// TIA Portal project "Perron038 AMR Siemens_2" (V14)

(* hardware
DEVICE "S7-1200 station_1"  S7-1200 Station
   slot 0: "Rack_0"  S7-1200 Rack  Rack  V1.0
   slot 1: "PLC_1"  CPU 1215C DC/DC/DC  6ES7 215-1AG40-0XB0  V4.2
*)

// ===== PLC "PLC_1"  CPU 1215C DC/DC/DC =====

VAR_GLOBAL   // PLC tag table "Default tag table"
   "Axis_1_Pulse" AT %Q0.0 : Bool;
   "Axis_1_Dir" AT %Q0.1 : Bool;
   "Axis_1_EN" AT %Q0.3 : Bool;
   "i_EndStopFWD" AT %I0.0 : Bool;
   "i_EndStopBWD" AT %I0.1 : Bool;
   "i_Switch8" AT %I0.7 : Bool;
   "i_Switch7" AT %I0.6 : Bool;
   "Servo_Pucks_Duration" AT %QW1002 : Int;
   "Servo_Grip_Duration" AT %QW1004 : Int;
   "System_Byte" AT %MB1 : Byte;
   "FirstScan" AT %M1.0 : Bool;
   "DiagStatusUpdate" AT %M1.1 : Bool;
   "AlwaysTRUE" AT %M1.2 : Bool;
   "AlwaysFALSE" AT %M1.3 : Bool;
   "Clock_Byte" AT %MB0 : Byte;
   "Clock_10Hz" AT %M0.0 : Bool;
   "Clock_5Hz" AT %M0.1 : Bool;
   "Clock_2.5Hz" AT %M0.2 : Bool;
   "Clock_2Hz" AT %M0.3 : Bool;
   "Clock_1.25Hz" AT %M0.4 : Bool;
   "Clock_1Hz" AT %M0.5 : Bool;
   "Clock_0.625Hz" AT %M0.6 : Bool;
   "Clock_0.5Hz" AT %M0.7 : Bool;
   "Tag_1" AT %Q0.2 : Bool;
   "Tag_2" AT %Q0.4 : Bool;
   "q_Lift_Up" AT %Q0.7 : Bool;
   "q_Lift_Down" AT %Q0.6 : Bool;
   "i_LiftDownStop" AT %I0.2 : Bool;
   "i_LiftHalte1" AT %I0.3 : Bool;
END_VAR

DATA_BLOCK "MotorControl_1_DB"   // DB1
{ S7_Optimized_Access := 'TRUE' }
VERSION : 0.1
// stored: InstanceOfName MotorControl_1
"MotorControl_1"
BEGIN
END_DATA_BLOCK

DATA_BLOCK "Horizontal_Movement_FB_DB"   // DB2
{ S7_Optimized_Access := 'TRUE' }
VERSION : 0.1
// stored: InstanceOfName Horizontal_Movement
"Horizontal_Movement"
BEGIN
END_DATA_BLOCK

DATA_BLOCK "ServoControl_1_DB"   // DB4
{ S7_Optimized_Access := 'TRUE' }
VERSION : 0.1
// stored: InstanceOfName ServoControl_Pucks
"ServoControl_Pucks"
BEGIN
END_DATA_BLOCK

DATA_BLOCK "ServoControl_2_DB"   // DB9
{ S7_Optimized_Access := 'TRUE' }
VERSION : 0.1
// stored: InstanceOfName ServoControl_Gripper
"ServoControl_Gripper"
BEGIN
END_DATA_BLOCK

DATA_BLOCK "DB_ModbusTCP_Connect"   // DB10
{ S7_Optimized_Access := 'TRUE' }
VERSION : 0.1
   VAR
      MBTCPClientRead : TCON_IP_v4;
      MBTCPClientRead_DISCONNECT : Bool;
      MBTCPClientRead_BUSY : Bool;
      MBTCPClientRead_ERROR : Bool;
      MBTCPClientRead_STATUS : Word;
   END_VAR
BEGIN
   MBTCPClientRead.InterfaceId := 64;
   MBTCPClientRead.ID := 16#1;
   MBTCPClientRead.ActiveEstablished := 1;
   MBTCPClientRead.RemoteAddress.ADDR[1] := 16#C0;
   MBTCPClientRead.RemoteAddress.ADDR[2] := 16#A8;
   MBTCPClientRead.RemoteAddress.ADDR[4] := 16#14;
   MBTCPClientRead.RemotePort := 502;
   MBTCPClientRead.LocalPort := 502;
   MBTCPClientRead.RemoteAddress.ADDR[3] := 16#C;
   MBTCPClientRead.ConnectionType := 16#B;
END_DATA_BLOCK

DATA_BLOCK "MBTCP_Data"   // DB11
{ S7_Optimized_Access := 'FALSE' }
VERSION : 0.1
   VAR
      Data : Array[1..1200] of Word;
   END_VAR
BEGIN
END_DATA_BLOCK

DATA_BLOCK "Noodstop_DB"   // DB12
{ S7_Optimized_Access := 'TRUE' }
VERSION : 0.1
// stored: InstanceOfName Noodstop
"Noodstop"
BEGIN
END_DATA_BLOCK

DATA_BLOCK "Lift_Control_DB"   // DB13
{ S7_Optimized_Access := 'TRUE' }
VERSION : 0.1
// stored: InstanceOfName Lift_Control
"Lift_Control"
BEGIN
END_DATA_BLOCK

DATA_BLOCK "Axis_1"   // DB3, Motion_DB
{ S7_Optimized_Access := 'TRUE' }
AUTHOR : SIMATIC
FAMILY : BasicMC
NAME : TO_PosAx
VERSION : 6.0
// stored: InstanceOfName TO_PositioningAxis
"TO_PositioningAxis"
BEGIN
   // Axis.HomingReferencePointSwitch_AddressCU = %I0.1
   // Axis.EnableOutput_AddressCU = %Q0.3
   // Axis.OnlinePtoModeCUEnumValue = PTO (pulse A and direction B)
   // Axis.OnlinePtoModeCU = 16#0000_0002
   // Axis.DirectionOutputEnabledCU = TRUE
   // Axis.SelectedChannel2EnumCU = %Q0.1
   // Axis.SelectedChannel1EnumCU = %Q0.0
   // Pulse.MinDeltaDeltaFrequencyCU = 0.004
   // Pulse.MaxDeltaDeltaFrequencyCU = 1.0E+10
   // Pulse.MinDeltaFrequencyCU = 0.005
   // Pulse.MaxDeltaFrequencyCU = 9.5E+9
   // Pulse.MinFrequencyCU = 1.0
   // Pulse.MaxFrequencyCU = 100000.0
   // Pulse.OutputSourceCU = 16#0000_0000
   // Axis.SelectPTO = 0
END_DATA_BLOCK

FUNCTION_BLOCK "MotorControl_1"   // FB1, SCL
{ S7_Optimized_Access := 'TRUE' }
VERSION : 0.1
   VAR_INPUT
      i_StartBWD : Bool;
      i_StartFWD : Bool;
      i_EndstopBWD : Bool;
      i_EndstopFWD : Bool;
   END_VAR
   VAR_OUTPUT
      q_mvFWD : Bool;
      q_mvBWD : Bool;
   END_VAR
BEGIN
   IF #i_StartBWD = TRUE THEN
       #q_mvBWD := 1;
   END_IF;

   IF #i_EndstopBWD = TRUE THEN
       #q_mvBWD := 0;
   END_IF;

   IF #i_StartFWD = TRUE THEN
       #q_mvFWD := 1;
   END_IF;

   IF #i_EndstopFWD = TRUE THEN
       #q_mvFWD := 0;
   END_IF;
END_FUNCTION_BLOCK

FUNCTION_BLOCK "ServoControl_Pucks"   // FB2, SCL
{ S7_Optimized_Access := 'TRUE' }
VERSION : 0.1
   VAR_INPUT
      "Modbus Data" : Array[1..1200] of Word;
   END_VAR
   VAR_OUTPUT
      PWM_Enable : Bool;
      q_ModbusMode : USInt;
      q_ModbusRequest : Bool;
   END_VAR
   VAR
      State : Int;
      TimerOnDelay : IEC_TIMER;
   END_VAR
BEGIN
   #PWM_Enable := 1;

   CASE #State OF
       0:
           #q_ModbusMode := 0;
           #q_ModbusRequest := 1;
           #State := 1;
           ;

       1:

           IF "MBTCP_Data".Data[4] = 16#0001 THEN
               #q_ModbusRequest := 0;
               #State := 2;
           ELSIF "MBTCP_Data".Data[4] = 16#0002 THEN
               #q_ModbusRequest := 0;
               #State := 3;
           END_IF;
           ;

       2:
           "Servo_Pucks_Duration" := 50;
           #State := 4;
       3:
           "Servo_Pucks_Duration" := 100;
           #State := 4;
       4:
           #q_ModbusRequest := 1;
           #State := 0;

       ELSE  // Statement section ELSE
           ;
   END_CASE;
END_FUNCTION_BLOCK

FUNCTION_BLOCK "Horizontal_Movement"   // FB3, SCL
{ S7_Optimized_Access := 'TRUE' }
VERSION : 0.1
   VAR_INPUT
      i_EstopFWD : Bool;
      i_EstopBWD : Bool;
      "Modbus Data" : Array[1..1200] of Word;
   END_VAR
   VAR_OUTPUT
      q_FWD : Bool;
      q_BWD : Bool;
      q_ModbusMode : USInt;
      q_ModbusRequest : Bool;
   END_VAR
   VAR
      State_HorMov : Int;
   END_VAR
BEGIN


   CASE #State_HorMov OF //Horizontale verplaatsing (max voor of achter)
           0:
           #q_ModbusMode := 0;
           #q_ModbusRequest := 1;
           #State_HorMov := 1;
           ;

           1:
           IF "MBTCP_Data".Data[2] = 16#0001 THEN
               #q_ModbusRequest := 0;
               #q_ModbusMode := 1;
               #State_HorMov := 2;
           ELSIF "MBTCP_Data".Data[2] = 16#0002 THEN
               #q_ModbusRequest := 0;
               #q_ModbusMode := 1;
               #State_HorMov := 3;
           END_IF;
           ;
       2:
           #q_FWD := 1;
           IF #i_EstopFWD THEN
               #q_FWD := 0;
               #State_HorMov := 4;
               ;
           END_IF;
       3:
           #q_BWD := 1;
           IF #i_EstopBWD THEN
               #q_BWD := 0;
               #State_HorMov := 4;
               ;
           END_IF;
           ;
       4:
           "MBTCP_Data".Data[2] := 16#0000;
           #q_ModbusRequest := 1;

           #State_HorMov := 0;
           ;
       ELSE  // Statement section ELSE
           ;
   END_CASE;
END_FUNCTION_BLOCK

FUNCTION_BLOCK "ServoControl_Gripper"   // FB4, SCL
{ S7_Optimized_Access := 'TRUE' }
VERSION : 0.1
   VAR_INPUT
      "Modbus Data" : Array[1..1200] of Word;
   END_VAR
   VAR_OUTPUT
      PWM_Enable : Bool;
      q_ModbusMode : USInt;
      q_ModbusRequest : Bool;
   END_VAR
   VAR
      State : Int;
      TimerOnDelay : IEC_TIMER;
   END_VAR
BEGIN
   #PWM_Enable := 1;

   CASE #State OF
       0:
           #q_ModbusMode := 0;
           #q_ModbusRequest := 1;
           #State := 1;
           ;

       1:

           IF "MBTCP_Data".Data[6] = 16#0001 THEN
               #q_ModbusRequest := 0;
               #State := 2;
           ELSIF "MBTCP_Data".Data[6] = 16#0002 THEN
               #q_ModbusRequest := 0;
               #State := 3;
           END_IF;
           ;

       2:
           "Servo_Grip_Duration" := 50;
           #State := 4;
       3:
           "Servo_Grip_Duration" := 100;
           #State := 4;
       4:
           #q_ModbusRequest := 1;
           #State := 0;

       ELSE  // Statement section ELSE
           ;
   END_CASE;
END_FUNCTION_BLOCK

FUNCTION_BLOCK "Lift_Control"   // FB5, SCL
{ S7_Optimized_Access := 'TRUE' }
VERSION : 0.1
   VAR_INPUT
      i_DownEnd : Bool;
      i_MidEnd1 : Bool;
   END_VAR
   VAR_OUTPUT
      q_Up : Bool;
      q_Down : Bool;
      q_ModbusMode : USInt;
      q_ModbusRequest : Bool;
   END_VAR
   VAR
      State : Int;
   END_VAR
BEGIN
   CASE #State OF
       0:
           #q_ModbusMode := 0;
           #q_ModbusRequest := 1;
           #State := 1;
           ;

       1:

           IF "MBTCP_Data".Data[8] = 16#0001 THEN
               #q_ModbusRequest := 0;
               #State := 2;
           ELSIF "MBTCP_Data".Data[8] = 16#0002 THEN
               #q_ModbusRequest := 0;
               #State := 3;
           ELSIF "MBTCP_Data".Data[8] = 16#0000 THEN
               #q_ModbusRequest := 0;
               #State := 4;
           ELSIF "MBTCP_Data".Data[8] = 16#0003 THEN
               #q_ModbusRequest := 0;
               #State := 5;
           END_IF;
           ;

       2:
           IF #i_DownEnd THEN
               #q_Down := 1;
               #q_Up := 0;
               #State := 6;

       ELSE
           #State := 6;
           #q_Down := 0;
       END_IF;
       3:
           #q_Down := 0;
           #q_Up := 1;
           #State := 6;
       4:
           #q_Down := 0;
           #q_Up := 0;
           #State := 6;

       5:
           IF #i_MidEnd1 THEN
               #q_Down := 0;
               #q_Up := 1;
               #State := 6;

           ELSE
               #State := 6;
               #q_Up := 0;
           END_IF;
       6:
           #q_ModbusRequest := 1;
           #State := 0;

       ELSE  // Statement section ELSE
           ;
   END_CASE;
END_FUNCTION_BLOCK

FUNCTION_BLOCK "Noodstop"   // FB6, SCL
{ S7_Optimized_Access := 'TRUE' }
VERSION : 0.1
   VAR_OUTPUT
      Lift1 : Bool;
      Lift2 : Bool;
      Motorcontrol : Bool;
      Motorcontrol2 : Bool;
   END_VAR
BEGIN
END_FUNCTION_BLOCK

FUNCTION "FC_MBTCP_Client" : Void   // FC10, LAD
{ S7_Optimized_Access := 'TRUE' }
VERSION : 0.1
   VAR_INPUT
      modbusmode : USInt;
      modbusrequest : Bool;
   END_VAR
BEGIN

REGION Network 1
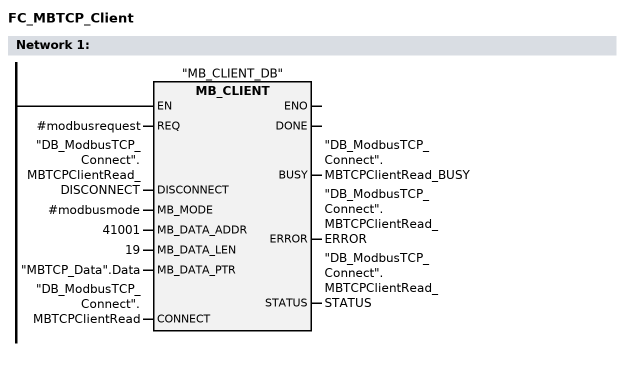
   "MB_CLIENT_DB"(REQ := #modbusrequest,   // MB_CLIENT
                  DISCONNECT := "DB_ModbusTCP_Connect".MBTCPClientRead_DISCONNECT,
                  MB_MODE := #modbusmode,
                  MB_DATA_ADDR := 41001,
                  MB_DATA_LEN := 19,
                  MB_DATA_PTR := "MBTCP_Data".Data,
                  CONNECT := "DB_ModbusTCP_Connect".MBTCPClientRead,
                  BUSY => "DB_ModbusTCP_Connect".MBTCPClientRead_BUSY,
                  ERROR => "DB_ModbusTCP_Connect".MBTCPClientRead_ERROR,
                  STATUS => "DB_ModbusTCP_Connect".MBTCPClientRead_STATUS);
END_REGION
END_FUNCTION

ORGANIZATION_BLOCK "Main"   // OB1, FBD, ProgramCycle
TITLE = "Main Program Sweep (Cycle)"
{ S7_Optimized_Access := 'TRUE' }
VERSION : 0.1
   VAR_INPUT
      Initial_Call : Bool;   // Initial call of this OB
      Remanence : Bool;   // =True, if remanent data are available
   END_VAR
   VAR_TEMP
      TimerReset : Bool;
      mvBtmp : Bool;
      mvFtmp : Bool;
      Gripper_Close : Bool;
      Gripper_Open : Bool;
      Pucks_Down : Bool;
      Pucks_Up : Bool;
      modbusModeTemp : USInt;
      modbusrequestTemp : Bool;
      PWMEnableServo1 : Bool;
      PWMEnableServo2 : Bool;
   END_VAR
BEGIN

REGION Network 1: Horizontal Movement
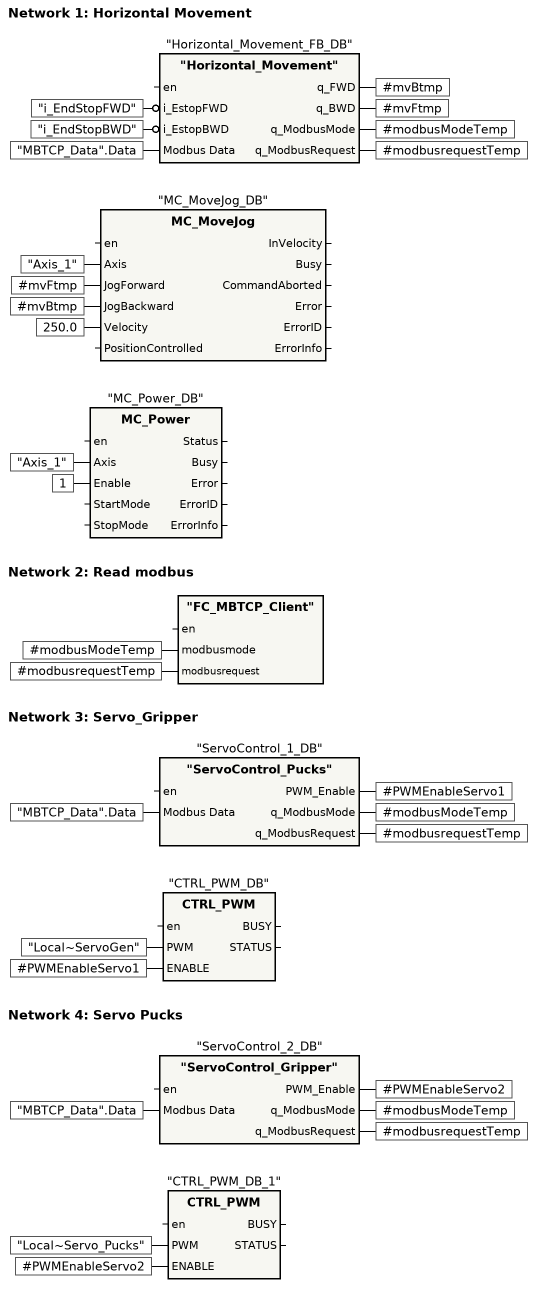
   "Horizontal_Movement_FB_DB"(i_EstopFWD := NOT "i_EndStopFWD",   // "Horizontal_Movement"
                           i_EstopBWD := NOT "i_EndStopBWD",
                           "Modbus Data" := "MBTCP_Data".Data,
                           q_FWD => #mvBtmp,
                           q_BWD => #mvFtmp,
                           q_ModbusMode => #modbusModeTemp,
                           q_ModbusRequest => #modbusrequestTemp);
   "MC_MoveJog_DB"(Axis := "Axis_1", JogForward := #mvFtmp, JogBackward := #mvBtmp, Velocity := 250.0);   // MC_MoveJog
   "MC_Power_DB"(Axis := "Axis_1", Enable := 1);   // MC_Power
END_REGION

REGION Network 2: Read modbus
   "FC_MBTCP_Client"(modbusmode := #modbusModeTemp, modbusrequest := #modbusrequestTemp);
END_REGION

REGION Network 3: Servo_Gripper
   "ServoControl_1_DB"("Modbus Data" := "MBTCP_Data".Data,   // "ServoControl_Pucks"
                       PWM_Enable => #PWMEnableServo1,
                       q_ModbusMode => #modbusModeTemp,
                       q_ModbusRequest => #modbusrequestTemp);
   "CTRL_PWM_DB"(PWM := "Local~ServoGen", ENABLE := #PWMEnableServo1);   // CTRL_PWM
END_REGION

REGION Network 4: Servo Pucks
   "ServoControl_2_DB"("Modbus Data" := "MBTCP_Data".Data,   // "ServoControl_Gripper"
                       PWM_Enable => #PWMEnableServo2,
                       q_ModbusMode => #modbusModeTemp,
                       q_ModbusRequest => #modbusrequestTemp);
   "CTRL_PWM_DB_1"(PWM := "Local~Servo_Pucks", ENABLE := #PWMEnableServo2);   // CTRL_PWM
END_REGION

REGION Network 5: Lift
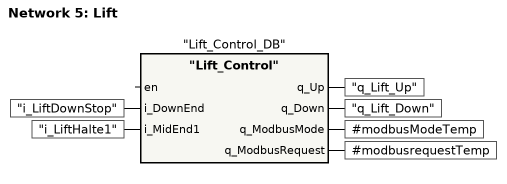
   "Lift_Control_DB"(i_DownEnd := "i_LiftDownStop",   // "Lift_Control"
                     i_MidEnd1 := "i_LiftHalte1",
                     q_Up => "q_Lift_Up",
                     q_Down => "q_Lift_Down",
                     q_ModbusMode => #modbusModeTemp,
                     q_ModbusRequest => #modbusrequestTemp);
END_REGION

REGION Network 6: Noodstop
END_REGION
END_ORGANIZATION_BLOCK